Yaskawa INFORM job: -1TEST.JBI

/JOB
//NAME -1TEST
//POS
///NPOS 2,0,0,0,0,0
///TOOL 0
///POSTYPE PULSE
///PULSE
C00000=-158986,58353,46093,126694,-152176,162476
C00001=-146791,60908,57910,117034,-155480,166998
//INST
///DATE 2018/11/08 16:29
///ATTR SC,RW
///GROUP1 RB1
NOP
MOVJ C00000 VJ=0.78
MOVJ C00001 VJ=0.78
END
